Universal Robots PolyScope program: gripper_tutorial.urp

Program gripper_tutorial (createdIn=3.3.0.0 lastSavedIn=3.5.2.10778 directory=/programs/usbdisk installation=default robotSerialNumber=2016352451)
Calibrated DH parameters: a=[0, -0.425, -0.39225, 0, 0, 0]; d=[0.089159, 0, 0, 0.10915, 0.09465, 0.0823]; alpha=[1.570796, 0, 0, 1.570796, -1.570796, 0]; deltaTheta=[0, 0, 0, 0, 0, 0]
Robot Program (runOnlyOnce=true motionType=MoveJ speed=1.047198 acceleration=1.396263 useActiveTCP=false)
  Popup Warning (haltProgram=false message=Don't modify this program. It will be erased at next boot.)
  'Activate the gripper before controlling it'
  Popup Message (haltProgram=false message=Activate the gripper before controling it)
  Script: rq_activate_and_wait()
  'Fully close the gripper and wait for completion'
  Popup Message (haltProgram=false message=Fully close the gripper and wait for completion)
  URCap Gripper (Robotiq_Grippers, Robotiq Inc.) dataModel(position=100, force=100, speed=79, blocking=true, positionInDouble=100.0, forceInDouble=100.0, speedInDouble=79.0)
  'Fully open the gripper and wait for completion'
  Popup Message (haltProgram=false message=Fully open the gripper and wait for completion)
  URCap Gripper (Robotiq_Grippers, Robotiq Inc.) dataModel(position=0, force=100, speed=79, blocking=true, positionInDouble=0.0, forceInDouble=100.0, speedInDouble=79.0)
  'Partially close the gripper and wait for completion'
  Popup Message (haltProgram=false message=Partially close the gripper and wait for completion)
  URCap Gripper (Robotiq_Grippers, Robotiq Inc.) dataModel(position=31, force=100, speed=79, blocking=true, positionInDouble=31.0, forceInDouble=100.0, speedInDouble=79.0)
  'Close the gripper and test the object detection'
  Popup Message (haltProgram=false message=Close the gripper and test the object detection)
  URCap Gripper (Robotiq_Grippers, Robotiq Inc.) dataModel(position=100, force=100, speed=79, blocking=true, positionInDouble=100.0, forceInDouble=100.0, speedInDouble=79.0)
  If rq_is_object_detected()
    'An object has been detected'
    Popup Message (haltProgram=false message=An object has been detected)
  Else 
    'No object detected'
    Popup Message (haltProgram=false message=No object detected)
  'Get the gripper current position in %. 100% is reached when the grippers is in encompassing mode.'
  Script: popup(rq_get_position(), "Gripper position (%)", blocking=True)
  'Command the gripper to open and continue the program execution.'
  Popup Message (haltProgram=false message=Command the gripper to open and continue the program execution.)
  URCap Gripper (Robotiq_Grippers, Robotiq Inc.) dataModel(position=0, force=0, speed=0, blocking=false, positionInDouble=0.0, forceInDouble=0.0, speedInDouble=0.0)
  'You can insert robot movement instructions while the gripper is moving'
  Wait Condition expression=rq_is_motion_complete()
  'Gripper motion completed'
  Popup Message (haltProgram=false message=Gripper motion completed)
  Folder Script Funtions
    Halt
    Folder Functions operating on a 0-100 span
      'Sets the gripper force [0-100]'
      Script: rq_set_force_norm(50)
      'Sets the gripper speed [0-100]'
      Script: rq_set_speed_norm(75)
      'Sends the partial move command and continue [0-100]'
      Script: rq_move_norm(75)
      'Sends the partial move command and wait until completion. [0-100]'
      Script: rq_move_and_wait_norm(30)
      'Sets the target position [0-100]'
      Script: rq_set_pos_norm(45)
      'Returns the gripper current position [0-100]'
      position := rq_current_pos_norm()
    Folder Functions operating on a 0-255 span
      'Sends the partial move command and wait until completion. [0-255]'
      Script: rq_move_and_wait(150)
      'Sets the target position'
      Script: rq_set_pos(150)
      'Returns the gripper current position [0-255]'
      position := rq_current_pos()
      'Sends the partial move command and continue'
      Script: rq_move(150)
      'Sets the gripper speed [0-255]'
      Script: rq_set_speed(255)
      'Sets the gripper force [0-255]'
      Script: rq_set_force(255)
    Folder Functions independant of the span
      'Activate the gripper if needed and wait for completion'
      Script: rq_activate_and_wait()
      'Activate the gripper and continue execution'
      Script: rq_activate()
      'Wait the end of activation'
      Wait Condition expression=rq_is_gripper_activated()
      'Sends the open command and continue'
      Script: rq_open()
      'Send the close command and continue'
      Script: rq_close()
      'Returns True if the motion is completed.'
      motion_complete := rq_is_motion_complete()
      'Returns True if an object has been detected.'
      object_detected := rq_is_object_detected()
      'Sends the open command and wait until completion'
      Script: rq_open_and_wait()
      'Sends the close command and wait until completion'
      Script: rq_close_and_wait()
      'Sets the goto bit to 1. Refer to user manual.'
      Script: rq_go_to()
      'Stops motion. The goto bit is cleared.'
      Script: rq_stop()
      'Sends the closing autorelease instruction and wait until completion'
      Script: rq_auto_release_close_and_wait()
      'Sends the opening autorelease instruction and wait until completion'
      Script: rq_auto_release_open_and_wait()
      'Resets the activation status of the gripper. Use after an autorelease before activating the gripper.'
      Script: rq_reset()
